TYPE DMC_Ins :
STRUCT
	DMC_Inputs : DriveInputs;
	DMC_POS_Status : PositionStatus;
	DMC_Drv_Status : DriveStatus;
END_STRUCT
END_TYPE

(* stored: Version 1.1.0.1, ProductVersion 3.1.4024.11
   DUT DMC_Ins: Id {8787cb22-c3a2-4ea4-a7f2-69f588a231f6} *)
